TYPE EMethod :
(
	MethGet := 1,
	MethPut := 2,
	MethResponse := 3
);
END_TYPE

(* stored: Version 1.1.0.1, ProductVersion 3.1.0.19
   DUT EMethod: Id {c5869327-cc50-4716-9d70-f7a091149913} *)
